PROGRAM HumidityPID
VAR
	
	PID: FB_BasicPID;
	bReset: BOOL;
	
	AH: LREAL;
	AHSetpoint: LREAL;
	
	//Constants for air as an ideal gas to calculate absolute humidity in g/m^3
	Tn:LREAL:=240.7263;
	m:LREAL:=7.591386;
	A:LREAL:=6.116441;
END_VAR

VAR_OUTPUT
	output: LREAL;
END_VAR

//Convert realative humidity to absolute humidity
AH:= A*EXPT	(10,m*GVL.Temp/(GVL.Temp+Tn))*(GVL.Humidity/100)*100*2.16679/(273.15+GVL.Temp);
AHSetpoint:= A*EXPT(10,m*GVL.TempSetpoint/(GVL.TempSetpoint+Tn))*(GVL.HumiditySetpoint/100)*100*2.16679/(273.15+GVL.TempSetpoint);

//Run pid loop
PID(
	fSetpointValue:=AHSetpoint,
	fActualValue:=AH, 
	bReset:=bReset, 
	fCtrlCycleTime:=1, 
	fKp:=1, 
	fTn:=1, 
	fTv:=1, 
	fTd:=0, 
	fCtrlOutput=>output);
	
	
//Since there's no dehumidification on this chamber
//Just reset the PID back to 0 if the output is negative
IF output<0 THEN
	output:=0;
	bReset:=TRUE;
ELSIF GVL.reset =  TRUE THEN
	bReset:=TRUE;
ELSE
	bReset:=FALSE;
END_IF

END_PROGRAM

(* stored: Version 1.1.0.1, ProductVersion 3.1.4022.16
   POU HumidityPID: Id {a8c07c7d-f9f1-49d5-818f-a19bd745ddbc}, SpecialFunc None *)
